// TIA Portal V17 export
FUNCTION "FC_BurnerAlarm" : Void   // FC, LAD
{ S7_Optimized_Access := 'TRUE' }
   VAR_TEMP   // added for the SCL form of the ladder/FBD networks
      _w1 : Bool;
      _w2 : Bool;
   END_VAR
BEGIN

REGION Network 1: 烧嘴故障报警置位蜂鸣器
   // 七个烧嘴故障反馈常开触点并联，汇总信号接入P_TRIG上升沿检测，任意故障反馈上升沿置位蜂鸣器输出。
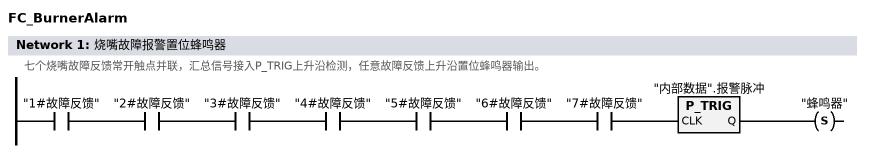
   RUNG wire#powerrail
      Contact( "1#故障反馈" )
      Contact( "2#故障反馈" )
      Contact( "3#故障反馈" )
      Contact( "4#故障反馈" )
      Contact( "5#故障反馈" )
      Contact( "6#故障反馈" )
      Contact( "7#故障反馈" )
      P_Trig( "内部数据".报警脉冲 )
      S_Coil( "蜂鸣器" )
   END_RUNG
   // the same network as SCL:
   #_w1 := "1#故障反馈" AND "2#故障反馈" AND "3#故障反馈" AND "4#故障反馈" AND "5#故障反馈" AND "6#故障反馈" AND "7#故障反馈";
   #_w2 := #_w1 AND NOT "内部数据".报警脉冲;   // rising edge
   "内部数据".报警脉冲 := #_w1;
   IF #_w2 THEN "蜂鸣器" := TRUE; END_IF;
END_REGION
END_FUNCTION
